// TIA Portal V20 export
DATA_BLOCK "DB_PressureLoop"   // DB6
{ S7_Optimized_Access := 'TRUE' }
VERSION : 0.1
// stored: AutoNumber true
BEGIN
END_DATA_BLOCK
